// TIA Portal V18 export
DATA_BLOCK "settingsSirene"   // DB25
{ S7_Optimized_Access := 'TRUE' }
VERSION : 0.1
// stored: AutoNumber false, DBAccessibleFromOPCUA true, DBAccessibleFromWebserver true, IsOnlyStoredInLoadMemory false, IsRetainMemResEnabled true, IsWriteProtectedInAS false, MemoryReserve 100, RetainMemoryReserve 100
   VAR RETAIN
      green { S7_SetPoint := 'True'} : "UDT_settingsSirene";
      yellow { S7_SetPoint := 'True'} : "UDT_settingsSirene";
      red { S7_SetPoint := 'True'} : "UDT_settingsSirene";
   END_VAR
BEGIN
END_DATA_BLOCK
